// TwinCAT 3 PLC project PRG_MachineSystem
// ProgramVersion: 3.1.4024.0
// CompilerDefines: VISU_USEWSTRING
// libraries:
//   B_Base, * (RafalOS)
//   B_HMIManager, * (RafałOS)
//   B_MachineControl, * (RafalOS)
//   B_MachineSystem, * (RafalOS)
//   Tc2_Standard, * (Beckhoff Automation GmbH)
//   Tc2_System, * (Beckhoff Automation GmbH)
//   Tc3_Module, * (Beckhoff Automation GmbH)
//   VisuSymbols,3.5.10.0,System
// project tree:
//   / DefaultInit.TcTTO, GlobalTextList.TcGTLO (not stored), MachineInit.TcTTO (not stored), PlcTask.TcTTO, Visualization Manager.TcVMO (not stored), VISU_TASK.TcTTO
//   GVLs/ GVL_MachineVariable.TcGVL
//   POUs/01_MachineConfiguration/ FB_MachineConfiguration.TcPOU
//   POUs/02_HMIConfiguration/ FB_HMIConfiguration.TcPOU
//   POUs/ PRG_MachineConfigure.TcPOU
//   VISUs/ MainScreen.TcVIS
// real-time tasks:
//   TASK PlcTask: cycle T#10ms, priority 10, ADS port 350
//   TASK VISU_TASK: cycle T#200000us, priority 12, ADS port 351
//   TASK DefaultInit: cycle T#10ms, priority 20, ADS port 352
//   TASK MachineInit: cycle T#10ms, priority 21, ADS port 353

CONFIGURATION PRG_MachineSystem
    RESOURCE PLC ON TwinCAT3
        TASK DefaultInit(INTERVAL := T#10ms, PRIORITY := 20);
        TASK PlcTask(INTERVAL := T#10ms, PRIORITY := 10);
        TASK VISU_TASK(INTERVAL := T#200000us, PRIORITY := 12);
        PROGRAM PRG_SystemControlMachineInit WITH DefaultInit : PRG_SystemControlMachineInit;
        PROGRAM PRG_SystemControlMachineWork WITH PlcTask : PRG_SystemControlMachineWork;
        PROGRAM VisuElems_Visu_Prg WITH VISU_TASK : VisuElems.Visu_Prg;
        PROGRAM PRG_ControlHMI WITH VISU_TASK : PRG_ControlHMI;
    END_RESOURCE
END_CONFIGURATION

// ---- GVLs/GVL_MachineVariable.TcGVL
{attribute 'qualified_only'}
VAR_GLOBAL
	fbMachineConfiguration		: FB_MachineConfiguration;
	fbHMIConfiguration			: FB_HMIConfiguration;
END_VAR

// ---- POUs/01_MachineConfiguration/FB_MachineConfiguration.TcPOU
(*			
	RafalOS
	Rafał Osajda		10.11.2025		TC 4024.66
	Główny blok konfiguracyjny MachineControl
*)
FUNCTION_BLOCK FB_MachineConfiguration EXTENDS FB_Base IMPLEMENTS ITF_MCConfiguration
VAR

END_VAR

METHOD AddHMIToMachineControl : BOOL
VAR_INPUT
	itfMachineControl			: ITF_MCMachineControlConfigure;
END_VAR
END_METHOD

METHOD PUBLIC AddTopElementToLogger : BOOL
VAR_INPUT
END_VAR
END_METHOD

(*			
	RafalOS
	Rafał Osajda		29.10.2025		TC 4024.66
	Dodawanie TopElementu do systemu
*)
METHOD PUBLIC AddTopElementToMachineControl : BOOL
VAR_INPUT
	itfMachineControl			: ITF_MCMachineControlConfigure;
END_VAR
END_METHOD

METHOD PUBLIC SetStartMode : BOOL
VAR_INPUT
	itfMachineControl			: ITF_MCMachineControlConfigure;
END_VAR
END_METHOD

METHOD StateAndModes : BOOL
VAR_INPUT
	itfMachineControl			: ITF_MCMachineControlConfigure;
END_VAR
END_METHOD

END_FUNCTION_BLOCK

// ---- POUs/02_HMIConfiguration/FB_HMIConfiguration.TcPOU
(*			
	RafalOS
	Rafał Osajda		10.11.2025		TC 4024.66
	Główny blok konfigurujący HMI
*)
FUNCTION_BLOCK FB_HMIConfiguration EXTENDS FB_Base IMPLEMENTS ITF_HMIConfiguration
VAR
END_VAR

END_FUNCTION_BLOCK

// ---- POUs/PRG_MachineConfigure.TcPOU
PROGRAM PRG_MachineConfigure
VAR
END_VAR

IF (NOT GVL_SystemVariable.bMachineInitDone) THEN

	IF (GVL_SystemVariable.itmpWywolanieMachineInit = 0) THEN
	GVL_SystemVariable.iLicznik	:= GVL_SystemVariable.iLicznik + 1;
	GVL_SystemVariable.itmpWywolanieMachineInit	:= GVL_SystemVariable.iLicznik;
	END_IF

	

	GVL_SystemVariable.fbMachineConfigure.AddConfiguration (fbConfigure := GVL_MachineVariable.fbMachineConfiguration);
	GVL_SystemVariable.fbHMIConfigure.AddConfiguration (fbConfigure := GVL_MachineVariable.fbHMIConfiguration);
	GVL_SystemVariable.bMachineInitDone		:= TRUE;
END_IF

END_PROGRAM

// ---- VISUs/MainScreen.TcVIS
VISUALIZATION MainScreen  // 2x2
END_VISUALIZATION
